GLOBALCONSTANTS Constants (* Global constants *)
  (* Standard: 61499-1 *)
  (* Version 1.0, 2025-12-21, franz *)
  PACKAGE OSCAT::Basic::Globals;
  IMPORT OSCAT::Basic::Data_types::CONSTANTS_MATH;
  VAR_GLOBAL CONSTANT
    MATH : OSCAT::Basic::Data_types::CONSTANTS_MATH;
  END_VAR
END_GLOBALCONSTANTS
